# EPICS autosave request: ioc/autoSaveRestore/sseq_settings.req
$(P)$(S).SCAN
$(P)$(S).DESC
$(P)$(S).PREC
$(P)$(S).DLY1
$(P)$(S).DOL1
$(P)$(S).DO1
$(P)$(S).STR1
$(P)$(S).LNK1
$(P)$(S).WAIT1
$(P)$(S).DLY2
$(P)$(S).DOL2
$(P)$(S).DO2
$(P)$(S).STR2
$(P)$(S).LNK2
$(P)$(S).WAIT2
$(P)$(S).DLY3
$(P)$(S).DOL3
$(P)$(S).DO3
$(P)$(S).STR3
$(P)$(S).LNK3
$(P)$(S).WAIT3
$(P)$(S).DLY4
$(P)$(S).DOL4
$(P)$(S).DO4
$(P)$(S).STR4
$(P)$(S).LNK4
$(P)$(S).WAIT4
